FUNCTION_BLOCK ACComponent EXTENDS ACObject IMPLEMENTS IACComponent
VAR_INPUT
END_VAR
VAR_OUTPUT
END_VAR
VAR
	_Childs : ARRAY [1..GCL.cChildsMAX] OF IACComponent;
	_Parent : IACComponent;
END_VAR

{attribute 'TcRpcEnable'}
PROPERTY ACIdentifier : STRING
GET
VAR
	i: INT;
	pos: INT;
END_VAR
pos := -1;
FOR i:=0 TO (LEN(_ACUrl) - 1) BY 1
  DO
  	//IF (_ACUrl[i] = '.') THEN
  	IF (_ACUrl[i] = 16#2E) THEN
		pos := i;
	END_IF
END_FOR;
IF (pos < 0) THEN
	ACIdentifier := '';
	RETURN;
END_IF
ACIdentifier := RIGHT(_ACUrl,LEN(_ACUrl) - pos + 1);
END_GET
END_PROPERTY

METHOD PROTECTED AddChild : BOOL
VAR_INPUT
	child : IACComponent;
END_VAR

VAR
	i: INT;
END_VAR
IF child = 0 THEN
	AddChild := FALSE;
	RETURN;
END_IF
// 1. Check if child already exists in the array because of online change
FOR i:=1 TO GCL.cChildsMAX BY 1
  DO
    IF _Childs[i] <> 0 THEN
		IF _Childs[i].ACUrl = child.ACUrl THEN
			AddChild := FALSE;
			RETURN;			
		END_IF
	ELSE
		EXIT;
	END_IF
END_FOR;
// 2. If the child doesn't exist, add to _Childs-List
FOR i:=1 TO GCL.cChildsMAX BY 1
  DO
    IF _Childs[i] = 0 THEN
		AddChild := TRUE;
		_Childs[i] := child;
		EXIT;
	END_IF
END_FOR;
END_METHOD

PROPERTY Childs : ARRAY [1..GCL.cChildsMAX] OF IACComponent
GET
Childs := _Childs;
END_GET
END_PROPERTY

METHOD PUBLIC FB_childinit
VAR_INPUT
END_VAR
VAR
	i: INT;
END_VAR
FOR i:=1 TO GCL.cChildsMAX BY 1
  DO
    IF _Childs[i] <> 0 THEN
		_Childs[i].FB_childinit();
	ELSE
		EXIT;
	END_IF
END_FOR;
END_METHOD

METHOD FB_init : BOOL
VAR_INPUT
	bInitRetains : BOOL; // if TRUE, the retain variables are initialized (warm start / cold start)
	bInCopyCode : BOOL;  // if TRUE, the instance afterwards gets moved into the copy code (online change)
	parent : IACComponent;
END_VAR

VAR
	isValidRef: BOOL;
END_VAR
IF parent <> 0 THEN
	_Parent := parent;
END_IF
IncFBInitCount();
END_METHOD

METHOD PUBLIC FB_postinit
VAR_INPUT
		root : IACVariobatch;
END_VAR
VAR
	i: INT;
END_VAR
SUPER^.FB_postinit(root);
FOR i:=1 TO GCL.cChildsMAX BY 1
  DO
    IF _Childs[i] <> 0 THEN
		_Childs[i].FB_postinit(root);
	ELSE
		EXIT;
	END_IF
END_FOR;
END_METHOD

METHOD FindChildOfTypeAt : IACComponent
VAR_INPUT
	atIndex : INT;
	objectType : TypeOfACObjectEnum;
	maxChildDepth : INT;
END_VAR
VAR
	currIndexInResultArr : INT;
	result : ARRAY [0..GCL.cChildsMAX] OF IACComponent;
END_VAR
currIndexInResultArr := 0;
FindChildsOfTypeIntern(THIS^,objectType,0,maxChildDepth,currIndexInResultArr,result);
FindChildOfTypeAt := result[atIndex];
END_METHOD

METHOD FindChildsOfType
VAR_INPUT
	objectType : TypeOfACObjectEnum;
	maxChildDepth : INT;
END_VAR
VAR_IN_OUT
	result : ARRAY [0..GCL.cChildsMAX] OF IACComponent;
END_VAR
VAR
	currIndexInResultArr : INT;
END_VAR
currIndexInResultArr := 0;
FindChildsOfTypeIntern(THIS^,objectType,0,maxChildDepth,currIndexInResultArr,result);
END_METHOD

METHOD PRIVATE FindChildsOfTypeIntern
VAR_INPUT
	iThis : IACComponent;
	objectType : TypeOfACObjectEnum;
	currentDepth : INT;
	maxChildDepth : INT;
END_VAR
VAR_IN_OUT
	currIndexInResultArr : INT;
	result : ARRAY [0..GCL.cChildsMAX] OF IACComponent;
END_VAR
VAR
	childs : ARRAY [1..GCL.cChildsMAX] OF IACComponent;
	i: INT;
	iProcessFunction : IPAProcessFunction;
	iDosing : IPAFDosing;
	iDischarging : IPAFDischarging;
	iMixing : IPAFMixing;
	
	iControlModule : IPAControlModule;
	iScaleBase : IPAScale;
	iScaleGravimetric : IPAScaleGravimetric;
	iScaleTotalizing : IPAScaleTotalizing;
	iScaleVolumetric : IPAScaleVolumetric;
	
	iProcessModule : IPAProcessModule;
	iSilo : IPAMSilo;
END_VAR
CASE objectType OF
	TypeOfACObjectEnum.ProcessFunction:
		IF __QUERYINTERFACE(iThis, iProcessFunction) THEN
			result[currIndexInResultArr] := iThis;
			currIndexInResultArr := currIndexInResultArr + 1;
		END_IF	
	TypeOfACObjectEnum.Dosing:
		IF __QUERYINTERFACE(iThis, iDosing) THEN
			result[currIndexInResultArr] := iThis;
			currIndexInResultArr := currIndexInResultArr + 1;
		END_IF	
	TypeOfACObjectEnum.Discharging:
		IF __QUERYINTERFACE(iThis, iDischarging) THEN
			result[currIndexInResultArr] := iThis;
			currIndexInResultArr := currIndexInResultArr + 1;
			RETURN;
		END_IF	
	TypeOfACObjectEnum.Mixing:
		IF __QUERYINTERFACE(iThis, iMixing) THEN
			result[currIndexInResultArr] := iThis;
			currIndexInResultArr := currIndexInResultArr + 1;
		END_IF	
	TypeOfACObjectEnum.ControlModule:
		IF __QUERYINTERFACE(iThis, iControlModule) THEN
			result[currIndexInResultArr] := iThis;
			currIndexInResultArr := currIndexInResultArr + 1;
		END_IF	
	TypeOfACObjectEnum.ScaleBase:
		IF __QUERYINTERFACE(iThis, iScaleBase) THEN
			result[currIndexInResultArr] := iThis;
			currIndexInResultArr := currIndexInResultArr + 1;
		END_IF	
	TypeOfACObjectEnum.ScaleGravimetric:
		IF __QUERYINTERFACE(iThis, iScaleGravimetric) THEN
			result[currIndexInResultArr] := iThis;
			currIndexInResultArr := currIndexInResultArr + 1;
		END_IF	
	TypeOfACObjectEnum.ScaleTotalizing:
		IF __QUERYINTERFACE(iThis, iScaleTotalizing) THEN
			result[currIndexInResultArr] := iThis;
			currIndexInResultArr := currIndexInResultArr + 1;
		END_IF	
	TypeOfACObjectEnum.ScaleVolumetric:
		IF __QUERYINTERFACE(iThis, iScaleVolumetric) THEN
			result[currIndexInResultArr] := iThis;
			currIndexInResultArr := currIndexInResultArr + 1;
		END_IF	
	TypeOfACObjectEnum.ProcessModule:
		IF __QUERYINTERFACE(iThis, iProcessModule) THEN
			result[currIndexInResultArr] := iThis;
			currIndexInResultArr := currIndexInResultArr + 1;
		END_IF	
	TypeOfACObjectEnum.Silo:
		IF __QUERYINTERFACE(iThis, iSilo) THEN
			result[currIndexInResultArr] := iThis;
			currIndexInResultArr := currIndexInResultArr + 1;
		END_IF	
END_CASE

IF currIndexInResultArr > GCL.cChildsMAX THEN
	RETURN;
END_IF
currentDepth := currentDepth + 1;
IF ((maxChildDepth > 0) AND (currentDepth > maxChildDepth)) THEN
	RETURN;
END_IF

childs := iThis.Childs;
FOR i:=1 TO GCL.cChildsMAX BY 1
  DO
    IF childs[i] <> 0 THEN
		FindChildsOfTypeIntern(childs[i],objectType,currentDepth,maxChildDepth,currIndexInResultArr,result);
	ELSE
		EXIT;
	END_IF
END_FOR;
END_METHOD

METHOD FindObjectByID : IACObject
VAR_INPUT
	instanceID	: UDINT;
END_VAR
VAR
	rootComp : IACComponent;
END_VAR
rootComp := Root;
IF rootComp = 0 THEN
	FindObjectByID := 0;
	RETURN;
END_IF
IF rootComp.InstanceID = instanceID THEN
	FindObjectByID := rootComp;
	RETURN;
END_IF
FindObjectByID := FindObjectInChilds(instanceID);
END_METHOD

METHOD PUBLIC FindObjectInChilds : IACObject
VAR_INPUT
	instanceID	: UDINT;
END_VAR
VAR
	i: INT;
	prevComponent : IACComponent;
	currentComponent : IACComponent;
END_VAR
prevComponent := 0;
currentComponent := 0;

FOR i:=1 TO GCL.cChildsMAX BY 1
  DO
    IF _Childs[i] <> 0 THEN
		currentComponent := _Childs[i];
		IF currentComponent.InstanceID = instanceID THEN
			FindObjectInChilds := currentComponent;
			RETURN;
		ELSIF currentComponent.InstanceID > instanceID THEN
			IF prevComponent <> 0 THEN
				FindObjectInChilds := prevComponent.FindObjectInChilds(instanceID);
				RETURN;
			ELSE
				FindObjectInChilds := 0;
				RETURN;
			END_IF
		ELSE
			prevComponent := currentComponent;
		END_IF
	ELSE
		EXIT;
	END_IF
END_FOR;

IF prevComponent <> 0 AND prevComponent.InstanceID < instanceID THEN
	FindObjectInChilds := prevComponent.FindObjectInChilds(instanceID);
	RETURN;
END_IF

FindObjectInChilds := 0;
END_METHOD

METHOD FindParentOfType : IACComponent
VAR_INPUT
	objectType : TypeOfACObjectEnum;
END_VAR
VAR
	iProcessFunction : IPAProcessFunction;
	iDosing : IPAFDosing;
	iDischarging : IPAFDischarging;
	iMixing : IPAFMixing;
	
	iControlModule : IPAControlModule;
	iScaleBase : IPAScale;
	iScaleGravimetric : IPAScaleGravimetric;
	iScaleTotalizing : IPAScaleTotalizing;
	iScaleVolumetric : IPAScaleVolumetric;
	
	iProcessModule : IPAProcessModule;
	iSilo : IPAMSilo;
END_VAR
IF objectType < TypeOfACObjectEnum.ProcessFunction OR _Parent = 0 THEN
	FindParentOfType := 0;
	RETURN;
END_IF

CASE objectType OF
	TypeOfACObjectEnum.ProcessFunction:
		IF __QUERYINTERFACE(_Parent, iProcessFunction) THEN
			FindParentOfType := _Parent;
			RETURN;
		END_IF	
	TypeOfACObjectEnum.Dosing:
		IF __QUERYINTERFACE(_Parent, iDosing) THEN
			FindParentOfType := _Parent;
			RETURN;
		END_IF	
	TypeOfACObjectEnum.Discharging:
		IF __QUERYINTERFACE(_Parent, iDischarging) THEN
			FindParentOfType := _Parent;
			RETURN;
		END_IF	
	TypeOfACObjectEnum.Mixing:
		IF __QUERYINTERFACE(_Parent, iMixing) THEN
			FindParentOfType := _Parent;
			RETURN;
		END_IF	
	TypeOfACObjectEnum.ControlModule:
		IF __QUERYINTERFACE(_Parent, iControlModule) THEN
			FindParentOfType := _Parent;
			RETURN;
		END_IF	
	TypeOfACObjectEnum.ScaleBase:
		IF __QUERYINTERFACE(_Parent, iScaleBase) THEN
			FindParentOfType := _Parent;
			RETURN;
		END_IF	
	TypeOfACObjectEnum.ScaleGravimetric:
		IF __QUERYINTERFACE(_Parent, iScaleGravimetric) THEN
			FindParentOfType := _Parent;
			RETURN;
		END_IF	
	TypeOfACObjectEnum.ScaleTotalizing:
		IF __QUERYINTERFACE(_Parent, iScaleTotalizing) THEN
			FindParentOfType := _Parent;
			RETURN;
		END_IF	
	TypeOfACObjectEnum.ScaleVolumetric:
		IF __QUERYINTERFACE(_Parent, iScaleVolumetric) THEN
			FindParentOfType := _Parent;
			RETURN;
		END_IF	
	TypeOfACObjectEnum.ProcessModule:
		IF __QUERYINTERFACE(_Parent, iProcessModule) THEN
			FindParentOfType := _Parent;
			RETURN;
		END_IF	
	TypeOfACObjectEnum.Silo:
		IF __QUERYINTERFACE(_Parent, iSilo) THEN
			FindParentOfType := _Parent;
			RETURN;
		END_IF	
END_CASE

FindParentOfType := _Parent.FindParentOfType(objectType);
END_METHOD

{attribute 'TcRpcEnable'}
METHOD PUBLIC InvokeSetterBool
VAR_INPUT
	PropertyID : INT;
	PropertyValue : BOOL;
END_VAR
END_METHOD

{attribute 'TcRpcEnable'}
METHOD PUBLIC InvokeSetterByte
VAR_INPUT
	PropertyID : INT;
	PropertyValue : BYTE;
END_VAR
END_METHOD

{attribute 'TcRpcEnable'}
METHOD PUBLIC InvokeSetterDInt
VAR_INPUT
	PropertyID : INT;
	PropertyValue : DINT;
END_VAR
END_METHOD

{attribute 'TcRpcEnable'}
METHOD PUBLIC InvokeSetterDT
VAR_INPUT
	PropertyID : INT;
	PropertyValue : DINT;
END_VAR
END_METHOD

{attribute 'TcRpcEnable'}
METHOD PUBLIC InvokeSetterEnum
VAR_INPUT
	PropertyID : INT;
	PropertyValue : INT;
END_VAR
END_METHOD

{attribute 'TcRpcEnable'}
METHOD PUBLIC InvokeSetterInt
VAR_INPUT
	PropertyID : INT;
	PropertyValue : INT;
END_VAR
END_METHOD

{attribute 'TcRpcEnable'}
METHOD PUBLIC InvokeSetterLReal
VAR_INPUT
	PropertyID : INT;
	PropertyValue : LREAL;
END_VAR
END_METHOD

{attribute 'TcRpcEnable'}
METHOD PUBLIC InvokeSetterReal
VAR_INPUT
	PropertyID : INT;
	PropertyValue : REAL;
END_VAR
END_METHOD

{attribute 'TcRpcEnable'}
METHOD PUBLIC InvokeSetterString
VAR_INPUT
	PropertyID : INT;
	PropertyValue : STRING;
END_VAR
END_METHOD

{attribute 'TcRpcEnable'}
METHOD PUBLIC InvokeSetterTime
VAR_INPUT
	PropertyID : INT;
	PropertyValue : DINT;
END_VAR
END_METHOD

{attribute 'TcRpcEnable'}
METHOD PUBLIC InvokeSetterUDInt
VAR_INPUT
	PropertyID : INT;
	PropertyValue : UDINT;
END_VAR
END_METHOD

{attribute 'TcRpcEnable'}
METHOD PUBLIC InvokeSetterUInt
VAR_INPUT
	PropertyID : INT;
	PropertyValue : UINT;
END_VAR
END_METHOD

METHOD PROTECTED OnMainEnter
VAR_INPUT
END_VAR
END_METHOD

METHOD PROTECTED OnMainExit
VAR_INPUT
END_VAR
END_METHOD

PROPERTY Parent : IACComponent
GET
Parent := _Parent;
END_GET
END_PROPERTY

PROPERTY Root : IACVariobatch
GET
VAR
	iVariobatch : IACVariobatch;
END_VAR
IF _Parent = 0 THEN
	IF __QUERYINTERFACE(THIS^, iVariobatch) THEN
		Root := iVariobatch;
	ELSE
		Root := 0;
	END_IF	
	RETURN;
END_IF
Root := _Parent.Root;
END_GET
END_PROPERTY

METHOD RunMain : BOOL
VAR
	i: INT;
END_VAR
OnMainEnter();
FOR i:=1 TO GCL.cChildsMAX BY 1
  DO
    IF _Childs[i] <> 0 THEN
		_Childs[i].RunMain();
	ELSE
		EXIT;
	END_IF
END_FOR;
OnMainExit();
END_METHOD

PROPERTY TypeOfACObject : TypeOfACObjectEnum
GET
TypeOfACObject := TypeOfACObjectEnum.Component;
END_GET
END_PROPERTY

END_FUNCTION_BLOCK

(* stored: Version 1.1.0.1, ProductVersion 3.1.4024.6
   POU ACComponent: Id {76279868-6a32-486d-b9cf-3518008e5244}, SpecialFunc None
   Property ACIdentifier: Id {5ae464c2-ab45-43ad-a768-ca043cd4b912}
   Get Get: Id {eec6f585-8237-47de-a6d7-45c5bba088db}
   Method AddChild: Id {ae80c3c5-eea9-4c65-9868-a7ea9cee5722}
   Property Childs: Id {bafde815-35f9-4ecf-8855-4c288fdc4e94}
   Get Get: Id {d18973ab-e112-4441-a434-734dad5bfb32}
   Method FB_childinit: Id {88990f67-0437-4b61-bd41-c32e91fff094}
   Method FB_init: Id {bd922afe-f463-416e-a54e-8a1973ea7698}
   Method FB_postinit: Id {eeb19e11-9936-4e16-bf7a-6d27ca54ca29}
   Method FindChildOfTypeAt: Id {6162b147-55dc-4849-82e2-51537856b6fb}
   Method FindChildsOfType: Id {cc966b9c-ebd0-4cbb-9495-ea40652f33e8}
   Method FindChildsOfTypeIntern: Id {b2bdf6ab-d225-4c7a-96f2-ec26236633f7}
   Method FindObjectByID: Id {414521d6-f4e8-4e3d-bb2e-5fb4f3102166}
   Method FindObjectInChilds: Id {22bbd2b5-21b6-47a1-a592-d1e51c460203}
   Method FindParentOfType: Id {6bef1b9e-3632-4c0a-a05c-0dce7580746f}
   Method InvokeSetterBool: Id {718df054-1fa9-4bbb-ade4-0f18ec834361}
   Method InvokeSetterByte: Id {0ae47c7b-e27c-4c57-88f8-1bc7082f5b03}
   Method InvokeSetterDInt: Id {6467ae74-c65c-4803-aae4-9b5feee2ae22}
   Method InvokeSetterDT: Id {073f28d0-0411-4390-9a52-128c857921f4}
   Method InvokeSetterEnum: Id {02198412-e73c-403e-963b-442e008a8c37}
   Method InvokeSetterInt: Id {02c64325-9090-4139-b762-3e63bb2acab6}
   Method InvokeSetterLReal: Id {a79e7c9a-95a0-4669-8e57-1dd82058e50f}
   Method InvokeSetterReal: Id {96ec4768-f738-4ba6-b9ed-010f2de59b2a}
   Method InvokeSetterString: Id {1cffcb77-44c5-4b33-b218-4342061684a0}
   Method InvokeSetterTime: Id {0bbf002b-6bdf-4695-9702-ad78cda90f14}
   Method InvokeSetterUDInt: Id {7386b95a-aff2-4eeb-8b3e-22f105ad1da4}
   Method InvokeSetterUInt: Id {218b7960-7982-45ce-a952-e36b6eb4aed2}
   Method OnMainEnter: Id {aa9c2f80-fd3a-4082-b6d7-1ae2308d1c9e}
   Method OnMainExit: Id {b5bb2bba-dd7c-4ecc-983c-59de5dff3d70}
   Property Parent: Id {613f2de5-844c-44e1-9d48-d7be61748a82}
   Get Get: Id {cae023ad-f08a-47e9-92ef-6d0ca88f1653}
   Property Root: Id {64fb832c-be64-4f35-ae48-b0115ce45b09}
   Get Get: Id {f0c1fbda-c5c9-4c3d-bb00-142367c24c43}
   Method RunMain: Id {77d1af51-fdbf-4046-bb5f-1017b9524e7e}
   Property TypeOfACObject: Id {e1f62ae0-634a-4888-a629-7fd887a0a2b7}
   Get Get: Id {4cf0edd4-eb86-457e-8bba-815fa32eff0c} *)
